# EPICS substitutions: timingApp/Db/timing.substitutions
file "perIOC.template"
{ pattern
{       T       P       R  }
  { "\$(T)" "\$(P)" "\$(R)" }
}

file "perTimingSequencer.template"
{ pattern
{       T     }
  { "\$(T)" }
}

file "perTimingSequencerVar.template"
{ pattern
{       T,               NAME,                     DESC }
  { "\$(T)", InjSeqSuccessCount,      "Number of successful non-default cycles" }
  { "\$(T)", InjSeqFailedCount,       "Number of failed non-default cycles" }
  { "\$(T)", InjSeqStartOverrunCount, "Count times that request came too late" }
  { "\$(T)", InjSeqDebug,             "Enable sequencer diagnostic messages" }
}
